PROGRAM MAIN
VAR
	stInstance : st_Event;
	bBoolean : BOOL := FALSE;
	RectangleA : FB_Rectangle;
	RectangleB : FB_Rectangle;
END_VAR

IF NOT bBoolean THEN
	UpdateEventTimeStampSystemTime (stEvent := stInstance);
	bBoolean := TRUE;
END_IF

END_PROGRAM

(* stored: Version 1.1.0.1, ProductVersion 3.1.4024.13
   POU MAIN: Id {a64fc99a-5ed5-44a8-a101-556d25ae14e7}, SpecialFunc None *)
